INTERFACE I_StateMachine

METHOD InnerLoopSM : BOOL
VAR_INPUT
END_VAR
END_METHOD

METHOD Reset : BOOL
VAR_INPUT
END_VAR
END_METHOD

METHOD Setup : BOOL
VAR_INPUT
END_VAR
END_METHOD

END_INTERFACE

(* stored: Version 1.1.0.1, ProductVersion 3.1.4024.12
   Itf I_StateMachine: Id {469cf387-cbed-4f2d-a0d7-5c52e983c171}
   Method InnerLoopSM: Id {8128a504-3343-4187-bad3-fc3e8ce0864e}
   Method Reset: Id {9f019809-cef4-4f8b-a231-5d682662cd0e}
   Method Setup: Id {adc45dd6-4d13-4542-9d3e-388be31631ca} *)
